{attribute 'qualified_only'}
{attribute 'strict'}
TYPE JsonErrors :
(
	enum_member := 0
);
END_TYPE

(* stored: Version 1.1.0.1, ProductVersion 3.1.4024.12
   DUT JsonErrors: Id {70782372-74d3-4ab2-984b-3680448a0838} *)
